// TIA Portal project "学习功能块FB" (V16)

(* hardware
DEVICE "S7-1200 station_1"  S7-1200 Station
   slot 0: "Rack_0"  S7-1200 Rack  Rack  V1.0
   slot 1: "PLC_1"  CPU 1214C DC/DC/Rly  6ES7 214-1HG40-0XB0  V4.4
*)

// ===== PLC "PLC_1"  CPU 1214C DC/DC/Rly =====

VAR_GLOBAL   // PLC tag table "默认变量表"
   "Tag_1" AT %I0.0 : Bool;
   "Tag_2" AT %I0.1 : Bool;
   "Tag_3" AT %Q0.0 : Bool;
   "Tag_4" AT %M0.0 : Bool;
   "Tag_5" AT %I1.0 : Bool;
   "Tag_6" AT %I1.1 : Bool;
   "Tag_7" AT %I1.2 : Bool;
   "Tag_8" AT %M0.1 : Bool;
   "Tag_9" AT %M0.2 : Bool;
END_VAR

DATA_BLOCK "队列_DB"   // DB1
{ S7_Optimized_Access := 'TRUE' }
VERSION : 0.1
// stored: InstanceOfName 队列
"队列"
BEGIN
END_DATA_BLOCK

FUNCTION_BLOCK "队列"   // FB1, LAD
{ S7_Optimized_Access := 'TRUE' }
VERSION : 0.1
   VAR_INPUT
      启动 : Bool;
      生成随机数 : Bool;
      踢出队列 : Bool;
      写入队列 : Bool;
      停止 : Bool;
   END_VAR
   VAR_OUTPUT
      运行标准位 : Bool;
      随机数 : UDInt;
      inter2 : UDInt;
   END_VAR
   VAR_IN_OUT
      程序步 : Bool;
   END_VAR
   VAR
      上一个周期3 : Bool;
      上一个周期2 : Bool;
      上一个周期1 : Bool;
      存储区 : Bool;
      日期 : DTL;
      inter : DInt;
      "ret——val" : Int;
      队列数组 : Array[0..9] of UDInt;
      数据缓存 : Array[0..9] of UDInt;
   END_VAR
   VAR CONSTANT
      "a" : Int := 20;
   END_VAR
   VAR_TEMP   // added for the SCL form of the ladder/FBD networks
      _w1 : Bool;
   END_VAR
BEGIN

REGION Network 1: 随机生成一个随机数
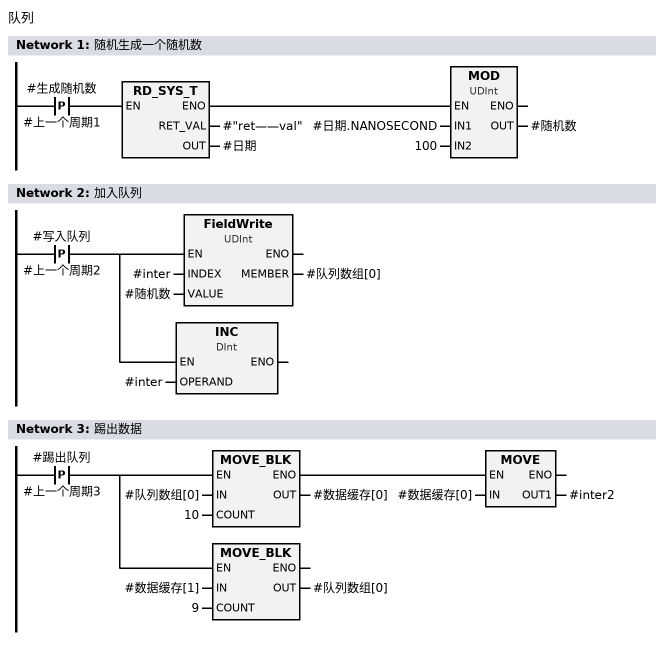
   // ENO of a box is taken as its EN; it also drops when the box reports an error
   #_w1 := #生成随机数 AND NOT #上一个周期1;   // rising edge of #生成随机数
   #上一个周期1 := #生成随机数;
   IF #_w1 THEN
       #"ret——val" := RD_SYS_T(OUT => #日期);
       #随机数 := #日期.NANOSECOND MOD 100;
   END_IF;
END_REGION

REGION Network 2: 加入队列
   // no SCL statement known for FieldWrite: written as a call
   #_w1 := #写入队列 AND NOT #上一个周期2;   // rising edge of #写入队列
   #上一个周期2 := #写入队列;
   IF #_w1 THEN
       FieldWrite(index := #inter, value := #随机数, member => #队列数组[0]);
       #inter := #inter + 1;
   END_IF;
END_REGION

REGION Network 3: 踢出数据
   #_w1 := #踢出队列 AND NOT #上一个周期3;   // rising edge of #踢出队列
   #上一个周期3 := #踢出队列;
   IF #_w1 THEN
       MOVE_BLK(IN := #队列数组[0], COUNT := 10, OUT => #数据缓存[0]);
       #inter2 := #数据缓存[0];
       MOVE_BLK(IN := #数据缓存[1], COUNT := 9, OUT => #队列数组[0]);
   END_IF;
END_REGION
END_FUNCTION_BLOCK

FUNCTION "MHJ-PLC-Lab-Function-S71200" : Void   // FC9000, SCL
{ S7_Optimized_Access := 'TRUE' }
VERSION : 0.1
   VAR_TEMP
      rdTimeReturn : Int;
      outputTime : DTL;
      SyncVal : Byte;
      forVal : Int;
      forVal_2 : Int;
      Value : Byte;
   END_VAR
   VAR CONSTANT
      CompVal : Byte := 16#34;
      Value_01 : Byte := 16#11;
      Value_01_DW : DWord := 16#A165_D992;
      Value_02_DW : DWord := 16#58BE_4401;
   END_VAR
BEGIN

   #Value:=PEEK(area := 16#82,
        dbNumber := 0,
        byteOffset := 511);
   #Value := #Value + 1;

   POKE(area := 16#82,
        dbNumber := 0,
        byteOffset := 511,
        value := #Value);

   POKE(area:=16#81,
        dbNumber:=0,
        byteOffset:=1016,
        value:=#Value_01_DW);
   POKE(area := 16#81,
        dbNumber := 0,
        byteOffset := 1020,
        value := #Value_02_DW);

   POKE(area := 16#81,
        dbNumber := 0,
        byteOffset := 511,
        value := B#16#00);

   FOR #forVal := 0 TO 120 DO
       FOR #forVal_2:=0 TO 10 DO
           #rdTimeReturn:=RD_SYS_T(#outputTime);
           #rdTimeReturn := WR_SYS_T(#outputTime);
           #rdTimeReturn := RD_SYS_T(#outputTime);
           #rdTimeReturn := WR_SYS_T(#outputTime);
       END_FOR;
       #SyncVal:= PEEK(area := 16#81,
                      dbNumber := 0,
                      byteOffset := 511);
       IF #SyncVal = #CompVal THEN
          GOTO M_1;
       END_IF;
   END_FOR;
   RETURN;

   M_1:
   POKE(area := 16#81,
        dbNumber := 0,
        byteOffset := 511,
        value := B#16#0);
END_FUNCTION

ORGANIZATION_BLOCK "Main"   // OB1, LAD, ProgramCycle
TITLE = "Main Program Sweep (Cycle)"
{ S7_Optimized_Access := 'TRUE' }
VERSION : 0.1
   VAR_INPUT
      Initial_Call : Bool;   // Initial call of this OB
      Remanence : Bool;   // =True, if remanent data are available
   END_VAR
BEGIN

REGION Network 1
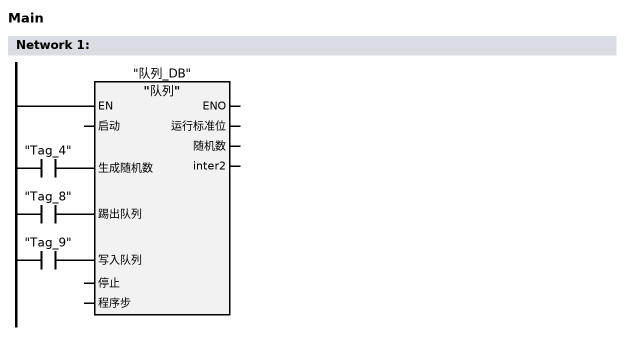
   RUNG wire#powerrail
      "队列_DB"(生成随机数 := wire#w1, 踢出队列 := wire#w2, 写入队列 := wire#w3, 启动 :=, 停止 :=, 程序步 :=, 运行标准位 =>, 随机数 =>, inter2 =>)
   END_RUNG
   RUNG wire#powerrail
      Contact( "Tag_4" )
   END_RUNG wire#w1
   RUNG wire#powerrail
      Contact( "Tag_8" )
   END_RUNG wire#w2
   RUNG wire#powerrail
      Contact( "Tag_9" )
   END_RUNG wire#w3
   // the same network as SCL:
   "队列_DB"(生成随机数 := "Tag_4", 踢出队列 := "Tag_8", 写入队列 := "Tag_9");   // "队列"
END_REGION
END_ORGANIZATION_BLOCK